// TwinCAT 3 PLC project PLC2
// ProgramVersion: 3.1.4026.1+c9eadab3edd020c56c333d811d5b3c408c2550c8
// libraries:
//   Tc2_Standard, * (Beckhoff Automation GmbH)
//   Tc2_System, * (Beckhoff Automation GmbH)
// project tree:
//   / PlcTask.TcTTO
//   POUs/ SecondPou.TcPOU, MAIN.TcPOU, FB_Singleton.TcPOU
// (motion and I/O tree: see PLC project plc1)
// real-time tasks:
//   TASK PlcTask1: cycle T#10ms, priority 21, ADS port 351
//   TASK PlcTask3: cycle T#10ms, priority 23, ADS port 353

CONFIGURATION PLC2
    RESOURCE PLC ON TwinCAT3
        TASK PlcTask(INTERVAL := T#10ms, PRIORITY := 23);
        PROGRAM MAIN WITH PlcTask : MAIN;
    END_RESOURCE
END_CONFIGURATION

// ---- POUs/MAIN.TcPOU
PROGRAM MAIN
VAR
	RealSingleton	: FB_Singleton;
	Singleton		: POINTER TO FB_Singleton;
	populate		: BOOL;
END_VAR

Singleton := RealSingleton.Instance;

IF populate THEN
	Singleton^.AddAlarm('Populated from main pou');
	populate := FALSE;
END_IF

SecondPou();

END_PROGRAM

// ---- POUs/FB_Singleton.TcPOU
{attribute 'enable_dynamic_creation'}
FUNCTION_BLOCK FB_Singleton
VAR
	_alarms 				: ARRAY[1..MAXNUMBEROFALRAMS] OF STRING;
	_actualNumberOfAlarms 	: UINT;
	_init 					: BOOL := FALSE;
END_VAR
VAR_STAT
	_instance 				: POINTER TO FB_Singleton := 0;
END_VAR
VAR CONSTANT
	MAXNUMBEROFALRAMS 		: UINT := 5;
END_VAR

METHOD AddAlarm : BOOL
VAR_INPUT
	message	: STRING;
END_VAR
IF _actualNumberOfAlarms <= MAXNUMBEROFALRAMS THEN
	_alarms[_actualNumberOfAlarms] := message;
	_actualNumberOfAlarms := _actualNumberOfAlarms + 1;
END_IF
END_METHOD

//FB_Exit must be implemented explicitly. If there is an implementation, then the
//method is called before the controller removes the code of the function block instance
//(implicit call). The return value is not evaluated.
METHOD FB_Exit: BOOL
VAR_INPUT
    bInCopyCode: BOOL;  // TRUE: the exit method is called in order to leave the instance which will be copied afterwards (online change).  
END_VAR
__DELETE(_instance);
END_METHOD

//FB_Init is always available implicitly and it is used primarily for initialization.
//The return value is not evaluated. For a specific influence, you can also declare the
//methods explicitly and provide additional code there with the standard initialization
//code. You can evaluate the return value.
METHOD FB_Init: BOOL
VAR_INPUT
    bInitRetains: BOOL; // TRUE: the retain variables are initialized (reset warm / reset cold)
    bInCopyCode: BOOL;  // TRUE: the instance will be copied to the copy code afterward (online change)   
END_VAR
IF NOT _init AND _instance = 0 THEN
	_instance := __NEW(FB_Singleton);
	_init := TRUE;
END_IF
_actualNumberOfAlarms := 1;
END_METHOD

PROPERTY Instance : POINTER TO FB_Singleton
GET
Instance := _instance;
END_GET
END_PROPERTY

END_FUNCTION_BLOCK

// ---- POUs/SecondPou.TcPOU
PROGRAM SecondPou
VAR
	RealSingleton	: FB_Singleton;
	Singleton		: POINTER TO FB_Singleton;
	populate		: BOOL;
END_VAR

Singleton := RealSingleton.Instance;

IF populate THEN
	Singleton^.AddAlarm('Populated from second pou');
	populate := FALSE;
END_IF

END_PROGRAM
